//set feed temperatures
hnhtControl.fFeedTemperature := fTargetTemperature_HNHT_Heating+localDefaultParameters.fOffset_FeedTemperature_HNHT;
hnltControl.fFeedTemperature_Heating := fTargetTemperature_HNLT_Heating+localDefaultParameters.fOffset_FeedTemperature_HNLT_Heating;
hnltControl.fFeedTemperature_Cooling := fTargetTemperature_HNLT_Cooling-localDefaultParameters.fOffset_FeedTemperature_HNLT_Cooling;
cnControl.fFeedTemperature := fTargetTemperature_CN-localDefaultParameters.fOffset_FeedTemperature_CN;
hnhtHnltLinkageControl.fFeedTemperature_HNHT := hnhtControl.fFeedTemperature;
hnhtHnltLinkageControl.fFeedTemperature_HNLT_Heating := hnltControl.fFeedTemperature_Heating;
hnhtHnltLinkageControl.fFeedTemperature_HNLT_Cooling := hnltControl.fFeedTemperature_Cooling;
hnltCnLinkageControl.fFeedTemperature_CN := cnControl.fFeedTemperature;
hnltCnLinkageControl.fFeedTemperature_HNLT_Heating := hnltControl.fFeedTemperature_Heating;
hnltCnLinkageControl.fFeedTemperature_HNLT_Cooling := hnltControl.fFeedTemperature_Cooling;

//set algorithm permission depending on production mode to control structs
CN_Check(fInput := cnState.fMidTemperature,
	fLowerLimit := aTemperatureLimits_CN[1],
	fUpperLimit := aTemperatureLimits_CN[2]);
cnControl.bAlgorithmPermission := CN_Check.bPermission;
	
HNLT_Check(fInput := hnltState.fMidTemperature,
	fLowerLimit := aTemperatureLimits_HNLT[1],
	fUpperLimit := aTemperatureLimits_HNLT[2]);
hnltControl.bAlgorithmPermission := HNLT_Check.bPermission;
	
HNHT_Check(fInput := hnhtState.fMidTemperature,
	fLowerLimit := aTemperatureLimits_HNHT[1],
	fUpperLimit := aTemperatureLimits_HNHT[2]);	
hnhtControl.bAlgorithmPermission := HNHT_Check.bPermission;
	
hnltCnLinkageControl.bAlgorithmPermission_CN := cnControl.bAlgorithmPermission;
hnltCnLinkageControl.bAlgorithmPermission_HNLT := hnltControl.bAlgorithmPermission;
hnhtHnltLinkageControl.bAlgorithmPermission_HNHT := hnhtControl.bAlgorithmPermission;
hnhtHnltLinkageControl.bAlgorithmPermission_HNLT := hnltControl.bAlgorithmPermission;
hnhtCnLinkageControl.bAlgorithmPermission_CN := cnControl.bAlgorithmPermission;
hnhtCnLinkageControl.bAlgorithmPermission_HNHT := hnhtControl.bAlgorithmPermission;
END_METHOD

END_FUNCTION_BLOCK

// ---- POUs/08 Lighting/FB_GA_Allgemein.TcPOU
FUNCTION_BLOCK FB_GA_Allgemein (*Setzt globale Parameter*)
VAR_INPUT
END_VAR
VAR_OUTPUT
END_VAR
VAR
	Uhrzeitgeber				: FB_CTRL_GET_SYSTEM_TIME;
	Uhrzeitgeber_Parameter	: ST_CTRL_GET_SYSTEM_TIME_PARAMS;
END_VAR

Uhrzeitgeber_Parameter.tTaskCycleTime	:= GA_Global.Zeit_TaskCycle;
Uhrzeitgeber_Parameter.tCtrlCycleTime	:= T#1m;

Uhrzeitgeber( stParams	:= Uhrzeitgeber_Parameter );

GA_Global.Systemzeit_Monat		:= WORD_TO_SINT(Uhrzeitgeber.stSystemTime.wMonth);
GA_Global.Systemzeit_Tag		:= WORD_TO_SINT(Uhrzeitgeber.stSystemTime.wDay);
GA_Global.Systemzeit_Wochentag	:= WORD_TO_SINT(Uhrzeitgeber.stSystemTime.wDayOfWeek);
GA_Global.Systemzeit_Stunde		:= WORD_TO_REAL(Uhrzeitgeber.stSystemTime.wHour) + WORD_TO_REAL(Uhrzeitgeber.stSystemTime.wMinute) / 60;

END_FUNCTION_BLOCK

// ---- POUs/08 Lighting/FB_Initialisierungsroutine.TcPOU
FUNCTION_BLOCK FB_Initialisierungsroutine
VAR_OUTPUT
END_VAR
VAR

END_VAR

(*Parameter System Beleuchtung *)
	Initialisierung.System_Bel_Parameter.AutoQuittierung := 0;
	Initialisierung.System_Bel_Parameter.Zeit_Vorl := 1000; (* Millisekunden *)
	Initialisierung.System_Bel_Parameter.Zeit_Nachl := 1000; (* Millisekunden *)
	Initialisierung.System_Bel_Parameter.Nachtabsenkung_Uhrzeit_Stunde_Start := 23; (*Uhr*)
	Initialisierung.System_Bel_Parameter.Nachtabsenkung_Uhrzeit_Stunde_Ende := 6; (*Uhr*)

END_FUNCTION_BLOCK

// ---- POUs/08 Lighting/Systeme/Sonstiges/Beleuchtung/Beleuchtung Außen/FB_System_BelAu_Logik.TcPOU
FUNCTION_BLOCK FB_System_BelAu_Logik
VAR_IN_OUT
	Steuerung	: ST_System_Bel_Steuerung;
	Zustand		: ST_System_Bel_Zustand;
END_VAR
VAR_INPUT
	Parameter	: ST_System_Bel_Parameter;
END_VAR
VAR_OUTPUT
END_VAR
VAR
END_VAR

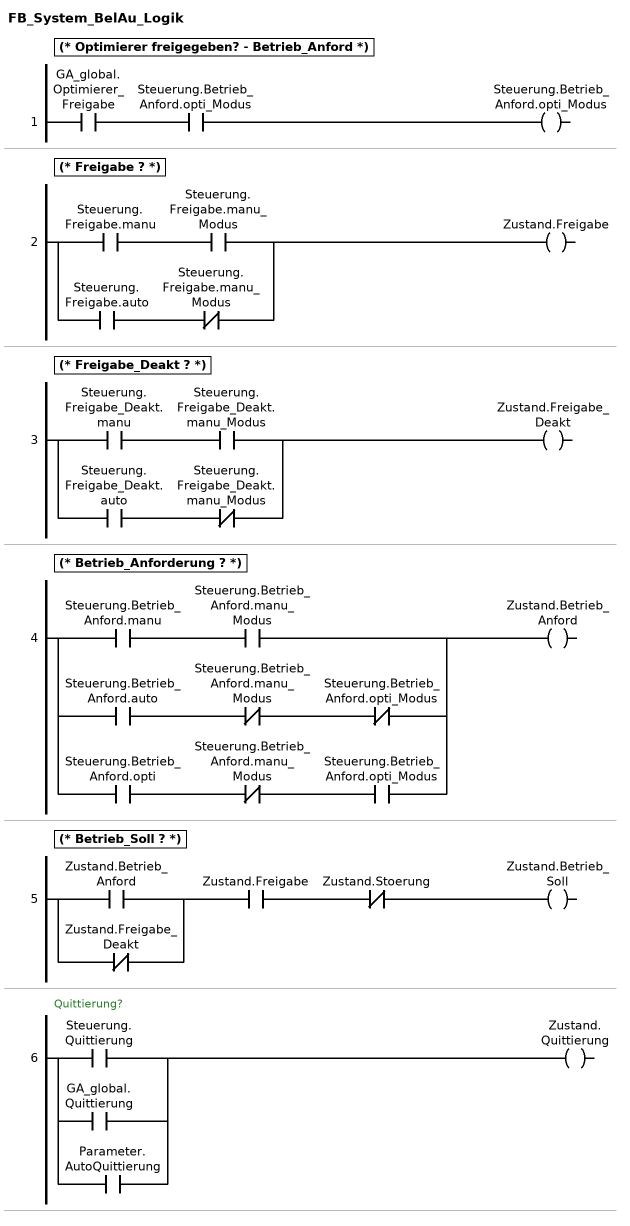
// NETWORK 1
// label: (* Optimierer freigegeben? - Betrieb_Anford *)
Steuerung.Betrieb_Anford.opti_Modus := GA_global.Optimierer_Freigabe AND Steuerung.Betrieb_Anford.opti_Modus;

// NETWORK 2
// label: (* Freigabe ? *)
Zustand.Freigabe := Steuerung.Freigabe.manu AND Steuerung.Freigabe.manu_Modus OR Steuerung.Freigabe.auto AND NOT Steuerung.Freigabe.manu_Modus;

// NETWORK 3
// label: (* Freigabe_Deakt ? *)
Zustand.Freigabe_Deakt := Steuerung.Freigabe_Deakt.manu AND Steuerung.Freigabe_Deakt.manu_Modus OR Steuerung.Freigabe_Deakt.auto AND NOT Steuerung.Freigabe_Deakt.manu_Modus;

// NETWORK 4
// label: (* Betrieb_Anforderung ? *)
Zustand.Betrieb_Anford := Steuerung.Betrieb_Anford.manu AND Steuerung.Betrieb_Anford.manu_Modus OR Steuerung.Betrieb_Anford.auto AND NOT Steuerung.Betrieb_Anford.manu_Modus AND NOT Steuerung.Betrieb_Anford.opti_Modus OR Steuerung.Betrieb_Anford.opti AND NOT Steuerung.Betrieb_Anford.manu_Modus AND Steuerung.Betrieb_Anford.opti_Modus;

// NETWORK 5
// label: (* Betrieb_Soll ? *)
Zustand.Betrieb_Soll := (Zustand.Betrieb_Anford OR NOT Zustand.Freigabe_Deakt) AND Zustand.Freigabe AND NOT Zustand.Stoerung;

// NETWORK 6
// Quittierung?
Zustand.Quittierung := Steuerung.Quittierung OR GA_global.Quittierung OR Parameter.AutoQuittierung;

END_FUNCTION_BLOCK

// ---- POUs/08 Lighting/Systeme/Sonstiges/Beleuchtung/Beleuchtung Außen/FB_System_BelAu_Regelung.TcPOU
FUNCTION_BLOCK FB_System_BelAu_Regelung
VAR_IN_OUT
	Stellwert					: ST_System_Bel_Stellwert;
	Steuerung					: ST_System_Bel_Steuerung;
	Zustand						: ST_System_Bel_Zustand;
END_VAR

VAR_INPUT

	Dunkelheits_Sensor_1			: REAL;

END_VAR
VAR_OUTPUT

	Steuerung_Farbcode_NO	: STRING;
	Steuerung_Farbcode_NW	: STRING;
	Steuerung_Farbcode_ND	: STRING;
	Steuerung_Farbcode_SO	: STRING;
	Steuerung_Farbcode_SW	: STRING;
	Steuerung_Farbcode_SD	: STRING;
END_VAR
VAR
	Dunkel: BOOL;
END_VAR

Dunkel:= FALSE;


IF Steuerung.Farbcode.manu_Modus THEN


	Stellwert.Leistung  := Zustand.Leistung;


	Steuerung_Farbcode_NO := Steuerung.Farbcode.manu;
	Steuerung_Farbcode_NW := Steuerung.Farbcode.manu;
	Steuerung_Farbcode_ND := Steuerung.Farbcode.manu;
	Steuerung_Farbcode_SO := Steuerung.Farbcode.manu;
	Steuerung_Farbcode_SW := Steuerung.Farbcode.manu;
	Steuerung_Farbcode_SD := Steuerung.Farbcode.manu;
ELSIF ( Dunkel AND NOT Steuerung.Farbcode.manu_Modus) THEN

	Stellwert.Leistung  := Zustand.Leistung;


	Steuerung_Farbcode_NO := Steuerung.Farbcode.auto;
	Steuerung_Farbcode_NW := Steuerung.Farbcode.auto;
	Steuerung_Farbcode_ND := Steuerung.Farbcode.auto;
	Steuerung_Farbcode_SO := Steuerung.Farbcode.auto;
	Steuerung_Farbcode_SW := Steuerung.Farbcode.auto;
	Steuerung_Farbcode_SD := Steuerung.Farbcode.auto;
ELSIF( NOT Dunkel AND NOT Steuerung.Farbcode.manu_Modus) THEN
Stellwert.Leistung  := Zustand.Leistung;


	Steuerung_Farbcode_NO := '000000';
	Steuerung_Farbcode_NW := '000000';
	Steuerung_Farbcode_ND := '000000';
	Steuerung_Farbcode_SO := '000000';
	Steuerung_Farbcode_SW := '000000';
	Steuerung_Farbcode_SD := '000000';

END_IF

END_FUNCTION_BLOCK

// ---- POUs/08 Lighting/Systeme/Sonstiges/Beleuchtung/Beleuchtung Außen/FB_System_BelAu_Sensorik.TcPOU
FUNCTION_BLOCK FB_System_BelAu_Sensorik
VAR_INPUT
END_VAR
VAR_OUTPUT
	(* Dunkelheit Sensor 1*)
	Dunkelheit_OUT	: REAL;
END_VAR
VAR
	(* Hardware oder DALI *)
	Dunkelheit_IN		: REAL;
END_VAR

(* ggfs Umrechung *)
Dunkelheit_OUT := Dunkelheit_IN * 3 ;

END_FUNCTION_BLOCK

// ---- POUs/08 Lighting/Systeme/Sonstiges/Beleuchtung/Beleuchtung Halle/FB_System_BelHa_Ablaufsteuerung.TcPOU
FUNCTION_BLOCK FB_System_BelHa_Ablaufsteuerung
VAR_IN_OUT
	Zustand			: ST_System_Bel_Zustand;
	Stellwert		: ST_System_Bel_Stellwert;
END_VAR
VAR_INPUT
	Steuerung		: ST_System_Bel_Steuerung;
	Parameter		: ST_System_Bel_Parameter;
END_VAR
VAR_OUTPUT
END_VAR
VAR
	Timer: TON;
END_VAR

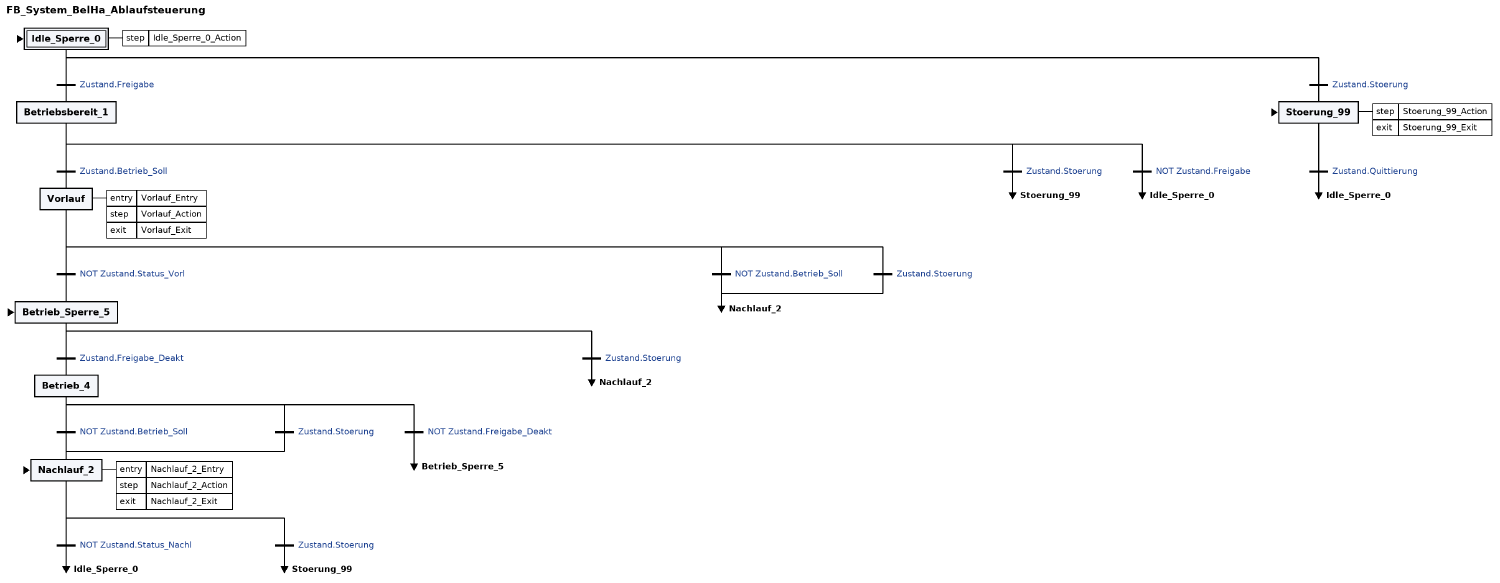
INITIAL_STEP Idle_Sperre_0:
    Idle_Sperre_0_Action(N);  // step action
END_STEP
TRANSITION FROM Idle_Sperre_0 TO Betriebsbereit_1
    := Zustand.Freigabe;
END_TRANSITION
TRANSITION FROM Idle_Sperre_0 TO Stoerung_99
    := Zustand.Stoerung;
END_TRANSITION
STEP Stoerung_99:
    Stoerung_99_Action(N);  // step action
    Stoerung_99_Exit(P0);  // exit action
END_STEP
TRANSITION FROM Stoerung_99 TO Idle_Sperre_0
    := Zustand.Quittierung;
END_TRANSITION
STEP Betriebsbereit_1:
END_STEP
TRANSITION FROM Betriebsbereit_1 TO Vorlauf
    := Zustand.Betrieb_Soll;
END_TRANSITION
TRANSITION FROM Betriebsbereit_1 TO Stoerung_99
    := Zustand.Stoerung;
END_TRANSITION
TRANSITION FROM Betriebsbereit_1 TO Idle_Sperre_0
    := NOT Zustand.Freigabe;
END_TRANSITION
STEP Vorlauf:
    Vorlauf_Entry(P1);  // entry action
    Vorlauf_Action(N);  // step action
    Vorlauf_Exit(P0);  // exit action
END_STEP
TRANSITION FROM Vorlauf TO Betrieb_Sperre_5
    := NOT Zustand.Status_Vorl;
END_TRANSITION
TRANSITION FROM Vorlauf TO Nachlauf_2
    := NOT Zustand.Betrieb_Soll;
END_TRANSITION
TRANSITION FROM Vorlauf TO Nachlauf_2
    := Zustand.Stoerung;
END_TRANSITION
STEP Betrieb_Sperre_5:
END_STEP
TRANSITION FROM Betrieb_Sperre_5 TO Betrieb_4
    := Zustand.Freigabe_Deakt;
END_TRANSITION
TRANSITION FROM Betrieb_Sperre_5 TO Nachlauf_2
    := Zustand.Stoerung;
END_TRANSITION
STEP Betrieb_4:
END_STEP
TRANSITION FROM Betrieb_4 TO Nachlauf_2
    := NOT Zustand.Betrieb_Soll;
END_TRANSITION
TRANSITION FROM Betrieb_4 TO Nachlauf_2
    := Zustand.Stoerung;
END_TRANSITION
TRANSITION FROM Betrieb_4 TO Betrieb_Sperre_5
    := NOT Zustand.Freigabe_Deakt;
END_TRANSITION
STEP Nachlauf_2:
    Nachlauf_2_Entry(P1);  // entry action
    Nachlauf_2_Action(N);  // step action
    Nachlauf_2_Exit(P0);  // exit action
END_STEP
TRANSITION FROM Nachlauf_2 TO Idle_Sperre_0
    := NOT Zustand.Status_Nachl;
END_TRANSITION
TRANSITION FROM Nachlauf_2 TO Stoerung_99
    := Zustand.Stoerung;
END_TRANSITION

ACTION Idle_Sperre_0_Action:
(* Quittierungszustand auf False setzen, damit das System bei einer erneuten Störung nicht direkt wieder angeschaltet wird *)
Steuerung.Quittierung	:= FALSE;
END_ACTION

ACTION Nachlauf_2_Action:
(* Nachlauf Timer starten *)
Timer( 	IN := Zustand.Status_Nachl,
		PT := DINT_TO_TIME(Parameter.Zeit_Nachl)
);
Zustand.Status_Nachl	:= NOT(Timer.Q AND NOT Zustand.Betrieb);

(* Stellwert setzen *)
Stellwert.Betrieb := FALSE;

(* Zustand setzen *)
Zustand.Status := E_Bel_Zustand_Status_Nachl;
END_ACTION

ACTION Nachlauf_2_Entry:
Zustand.Status_Nachl := TRUE;
(* Reset Timer *)
Timer(IN := FALSE);
END_ACTION

ACTION Nachlauf_2_Exit:
Zustand.Status_Nachl := FALSE;
END_ACTION

ACTION Stoerung_99_Action:
(* Stellwert setzen *)
Stellwert.Betrieb := FALSE;

(* Zustand setzen *)
Zustand.Stoerung := TRUE;
Zustand.Status := E_Bel_Zustand_Status_Stoerung;
END_ACTION

ACTION Stoerung_99_Exit:
Zustand.Stoerung	:= FALSE;
END_ACTION

ACTION Vorlauf_Action:
(* Vorlaufzeit Timer starten *)
Timer( 	IN := Zustand.Status_Vorl,
		PT := DINT_TO_TIME(Parameter.Zeit_Vorl)
);
Zustand.Status_Vorl := NOT (Timer.Q AND Zustand.Betrieb);

(* Stellwert setzen *)
Stellwert.Betrieb 	:= TRUE;
Stellwert.Leistung  := Zustand.Leistung;
(* Zustand setzen *)
Zustand.Status := E_Bel_Zustand_Status_Vorl;
END_ACTION

ACTION Vorlauf_Entry:
Zustand.Status_Vorl := TRUE;
(* Reset Timer *)
Timer(IN := FALSE);
END_ACTION

ACTION Vorlauf_Exit:
Zustand.Status_Vorl := FALSE;
END_ACTION

END_FUNCTION_BLOCK

// ---- POUs/08 Lighting/Systeme/Sonstiges/Beleuchtung/Beleuchtung Halle/FB_System_BelHa_Sensorik.TcPOU
FUNCTION_BLOCK FB_System_BelHa_Sensorik
VAR_INPUT
END_VAR
VAR_OUTPUT
	(* Helligkeit Sensor 1*)
	HelligkeitSensor_1_OUT	: REAL;
	HelligkeitSensor_2_OUT	: REAL;
	(* Helligkeit Sensor 2*)
END_VAR
VAR
	(* Hardware oder DALI *)
	SensorHalle1				: FB_Bel_Lichtsensor;
	HelligkeitSensor_1_IN		: REAL;
	HelligkeitSensor_2_IN		: REAL;
END_VAR

(* ggfs Umrechung *)
HelligkeitSensor_1_OUT := HelligkeitSensor_1_IN * 3 ;
HelligkeitSensor_2_OUT := HelligkeitSensor_2_IN * 3;

END_FUNCTION_BLOCK

// ---- POUs/08 Lighting/Systeme/Sonstiges/Beleuchtung/Beleuchtung Halle/FB_System_BelHa_Stellwertscheck.TcPOU
FUNCTION_BLOCK FB_System_BelHa_Stellwertscheck
VAR_IN_OUT
	Stellwert	: ST_System_Bel_Stellwert;
END_VAR

VAR_INPUT
	Zustand		: ST_System_Bel_Zustand;
	Parameter	: ST_System_Bel_Parameter;
END_VAR
VAR_OUTPUT
END_VAR
VAR
END_VAR

Stellwert.Leistung  := Zustand.Leistung;

IF( Stellwert.Betrieb ) THEN
	CASE Zustand.Regelung_Modus OF
		E_Bel_Regelung_Modus_P:	(* Steuerung durch Taster *)
			(* Max-Min-Grenzen erzwingen *)
			Stellwert.Leistung	 := MIN(Parameter.Stellwert_Leistung_max, Stellwert.Leistung);
			Stellwert.Leistung	 := MAX(Parameter.Stellwert_Leistung_min, Stellwert.Leistung);

		E_Bel_Regelung_Modus_Lichtsensor:	(* Regelung durch Lichtsensor *)
			(* Max-Min-Grenzen erzwingen *)
			Stellwert.Leistung		 := MIN(Parameter.Stellwert_Leistung_max, Stellwert.Leistung);
			Stellwert.Leistung		 := MAX(Parameter.Stellwert_Leistung_min, Stellwert.Leistung);

ELSE
		Stellwert.Leistung	:= 0;
	END_CASE;
ELSE
	Stellwert.Leistung	:= 0;
END_IF;

END_FUNCTION_BLOCK

// ---- POUs/08 Lighting/Systeme/Sonstiges/Beleuchtung/Beleuchtung Halle/FB_System_BelHa_Zustandscheck.TcPOU
FUNCTION_BLOCK FB_System_BelHa_Zustandscheck
VAR_IN_OUT
	Zustand					: ST_System_Bel_Zustand;
END_VAR
VAR_INPUT
	Steuerung				: ST_System_Bel_Steuerung;
	Parameter				: ST_System_Bel_Parameter;
END_VAR
VAR_OUTPUT
END_VAR
VAR
	Timer1: TON;
	Timer2: TON;
END_VAR

(*
	Stoerung_Code
		0:	*Allgemein Störung Beleuchtung (intern)
		1:	* Störung durch DALI-Lib
		2:	..
		3:
		4:
		5:
		6:
		7:

	Warnung_Code
		0:	*Allgemein Warnung Beleuchtung (intern)
		1:	keine Betriebsrückmeldung
		2:	keine Leistung
		3:	*Beleuchtung im Handbetrieb
		4:
		5:
		6:
		7:

	Freigabe_Code
		0:	*Freigabe durch Automatik entzogen
		1:	*Freigabe durch Manuell entzogen
		2:	*Freigabe durch Stoerung entzogen
		3: 	*Freigabe durch hohe Einschalthäufigkeiten entzogen
		4: 	*Freigabe durch zu hohe Rücklauf-Temperaturen entzogen
*)
(* Zustandsdefinitionen *)
Zustand.Betrieb	:= zustand.Betrieb_Anford AND Zustand.Freigabe  ;



Timer1(	IN := (Zustand.Betrieb_Anford <> Zustand.Betrieb),
		PT := T#1M,
		Q => Zustand.Warnung_Code.1
);

(* Warnung - keine Leistung im Betrieb nach 1 Minute *)
Timer2(	IN := Zustand.Leistung <= 0 AND Zustand.Betrieb_Anford = TRUE,
		PT := T#1M,
		Q => Zustand.Warnung_Code.2
);

END_FUNCTION_BLOCK

// ---- POUs/08 Lighting/Systeme/Sonstiges/Beleuchtung/FB_Beleuchtung.TcPOU
FUNCTION_BLOCK FB_Beleuchtung
VAR_INPUT
END_VAR
VAR_OUTPUT
END_VAR
VAR
	Hallenbeleuchtung: FB_System_BelHa;
	Aussenbeleuchtung: FB_System_BelAu;
END_VAR

Hallenbeleuchtung(Freigabe_auto := TRUE, Betrieb_Anford_auto := TRUE, AdressType := eDALIV2AddrTypeGroup); // FB_System_BelHa
Aussenbeleuchtung(Freigabe_auto := TRUE, Betrieb_Anford_auto := TRUE, AdressType := eDALIV2AddrTypeGroup); // FB_System_BelAu

END_FUNCTION_BLOCK
